Staubli VAL3: onBackEvent.pgx

program onBackEvent(bool& x_bSave[])
  local num i
  local string l_sMessage[3]
  local num l_nLocal
  local bool l_bYes
  local string l_sAction[3]
  local num l_nIndex
  local string l_sButton[2]
begin

end
